// Brief: Slave Arm move to Package posture
FUNCTION_BLOCK PUBLIC FB_SlaveCtrlPackage EXTENDS FB_SlaveArmCtrlBase
VAR_INPUT
END_VAR
VAR_OUTPUT
END_VAR
VAR
	// packageDHJntPos
	m_packageJntPosSlave :Vec8d := 	[0.0, 1.13-pi/2, 0.535, 0, 0, 0, 0, 0];
	m_packageMaxJntVel: Vec8d := [2(20*g_deg2Rad), 0.05, 5(20*g_deg2Rad)];
	m_packageMaxJntAcc: Vec8d := [2(40*g_deg2Rad), 0.1, 5(40*g_deg2Rad)];
	m_packageMaxJntJerk: Vec8d := [2(80*g_deg2Rad),0.4, 5(80*g_deg2Rad)];
	
	m_jntVelFilt :ARRAY[1..3] OF FB_LowPassFilter;
	
	m_endJntPos:Vec8d;
	m_packageMotionKp :LREAL := 10;
END_VAR

// override this function in each exact controller
METHOD PROTECTED calcCmdJntPos : BOOL
VAR_IN_OUT CONSTANT
	// endoscope pose in cart coordinate
	i_endoscopePose : ST_Frame;
	
	// master arm data
	i_masterStatus :ST_MasterStatus;
	
	// setup arm data
	i_setupStatus: ST_SetupStatus;
	
	// slave arm data
	i_slaveArm :FB_SlaveArm;
END_VAR

VAR 
	i :INT;
	curJntPos, posErr :Vec8d;
	collisionAvoidJntVel:Vec2d;
END_VAR
// package motino
FOR i:=1 TO 3 DO 
	m_cmdJntVel[i] := m_packageMotionKp *(m_endJntPos[i]-m_cmdJntPos[i]);
	m_cmdJntVel[i] := LIMIT(-m_packageMaxJntVel[i], m_cmdJntVel[i], m_packageMaxJntVel[i]);
END_FOR

// self-collision avoid velocity
collisionAvoidJntVel:=i_slaveArm.m_repulseJntVel;

FOR i:=1 TO 3 DO 
	IF i<3 THEN
		m_cmdJntVel[i]:=m_jntVelFilt[i].run(m_cmdJntVel[i]+collisionAvoidJntVel[i]);
	ELSE
		m_cmdJntVel[i]:=m_jntVelFilt[i].run(m_cmdJntVel[i]);
	END_IF
	
	// boundary limit
	IF (m_cmdJntPos[i] > GVL_SlaveMotorParameters.g_maxDHJntPos[i] AND m_cmdJntVel[i] > 0) OR
		(m_cmdJntPos[i] < GVL_SlaveMotorParameters.g_minDHJntPos[i] AND m_cmdJntVel[i] < 0) THEN
		m_cmdJntVel[i] :=0;
	END_IF
	
	m_cmdJntPos[i] := m_cmdJntPos[i] + m_cmdJntVel[i] * g_slaveArmCtrlCycleTime;
END_FOR

// check IF TO terminate
curJntPos := i_slaveArm.curJntPos;
vecSub(m_packageJntPosSlave, curJntPos, posErr);
m_isFinished :=ABS(posErr[1])<g_jntCtrlAngTolLow AND ABS(posErr[2])<g_jntCtrlAngTolLow AND ABS(posErr[3])<g_cartCtrlPosTolLow;
END_METHOD

METHOD PUBLIC init : BOOL
VAR_IN_OUT CONSTANT
	i_slaveArm	:FB_SlaveArm;
END_VAR
VAR_IN_OUT 
	r_slaveArmCtrlCmd :ST_SlaveArmCtrlCmds;
END_VAR

VAR
	i :INT;
	startJntPos,endJntPos :Vec8d;
END_VAR
// check if to hold the command joint position unchanged
m_holdLastCmds := checkToHoldLastCmds(i_slaveArm);

//init
SUPER^.Init(i_slaveArm,r_slaveArmCtrlCmd);
m_packageJntPosSlave[3] := GVL_SlaveMotorParameters.g_maxDHJntPos[3];

//traj plan
startJntPos:= i_slaveArm.curJntPos;
endJntPos := i_slaveArm.curJntPos;
FOR i := 1 TO 3 DO
	endJntPos[i] := m_packageJntPosSlave[i];
END_FOR
m_endJntPos:=endJntPos;

FOR i:=1 TO 3 DO
	m_jntVelFilt[i].init(1, 1, g_slaveArmCtrlFreq);
	m_jntVelFilt[i].run(0);
END_FOR



// update commands to arm
copyCmds(r_slaveArmCtrlCmd);
END_METHOD

END_FUNCTION_BLOCK

(* stored: Version 1.1.0.1, ProductVersion 3.1.4024.11
   POU FB_SlaveCtrlPackage: Id {f1b722f8-ced5-4c88-9461-cc1a45d6acc0}, SpecialFunc None
   Method calcCmdJntPos: Id {5a4931eb-3ea0-408d-a661-3a3f375fd93d}
   Method init: Id {b23724e4-deb7-4c43-8ea2-717cb3ca8f89} *)
